{attribute 'qualified_only'}
{attribute 'strict'}
TYPE E_MachineState :
(
	IDLE := 0,
	WAIT_FOR_BOTTLE,
	FILLING,
	COMPLETED,
	STOPPED,
	ERROR
);
END_TYPE

(* stored: Version 1.1.0.1, ProductVersion 3.1.4024.16
   DUT E_MachineState: Id {a719bc55-830b-4b24-bab3-0045d5a36331} *)
